// TIA Portal V20 export
TYPE "LER_typeRadiusMeasureCommnads"
// stored: Access Published
   STRUCT
      ZeroSet : Bool;
      Reset : Bool;
   END_STRUCT;
END_TYPE
